PROGRAM PRG_LVCP5_Group3
VAR
    // Function Block Instance
    fbContactor: FB_ContactorControl;

    // Contactor 1 IO Structure  
    stContactor_IO: ST_ContactorIO;
    
    // Başlangıç konfigürasyonu için flag
    bContactorInitDone: BOOL := FALSE;
    bCapacitorInitDone: BOOL := FALSE;	
END_VAR



	M_Contactor();
	
	M_Capacitor();

METHOD M_Capacitor : BOOL
VAR
    nGroupIndex : INT;
END_VAR

nGroupIndex := 2;  // Grup 3 için index

IF NOT bCapacitorInitDone THEN
    // Grup 3 değerlerini ata
    GVL_LVCP5.astCompensationGroups[nGroupIndex].rPower := 10.0;
    GVL_LVCP5.astCompensationGroups[nGroupIndex].rVoltage := 450.0;
    GVL_LVCP5.astCompensationGroups[nGroupIndex].nQuantity := 8;
    GVL_LVCP5.astCompensationGroups[nGroupIndex].sTagPrefix := '+EP8-22C1';
    GVL_LVCP5.astCompensationGroups[nGroupIndex].sProductCode := 'ENT.CXD-450-10';
    
    bCapacitorInitDone := TRUE;
END_IF

// Grup 3 aktif durumu
GVL_LVCP5.abGroupActive[nGroupIndex] := stContactor_IO.bFeedback;

M_Capacitor := TRUE;
END_METHOD

METHOD M_Contactor : BOOL
VAR_INPUT
END_VAR
IF NOT bContactorInitDone THEN
    // Konfigürasyon parametreleri
    GVL_LVCP5.stGroup3_ContactorHMI.stConfig.sProjectCode := '+EP8-23K1';
    GVL_LVCP5.stGroup3_ContactorHMI.stConfig.sProductCode := 'SCH LC1G185LSEA';
    GVL_LVCP5.stGroup3_ContactorHMI.stConfig.rRatedCurrent := 185.0;
    GVL_LVCP5.stGroup3_ContactorHMI.stConfig.rRatedVoltage := 1000.0;
    GVL_LVCP5.stGroup3_ContactorHMI.stConfig.nPhaseCount := 3;
    GVL_LVCP5.stGroup3_ContactorHMI.stConfig.tFeedbackDelay := T#500MS;
    GVL_LVCP5.stGroup3_ContactorHMI.stConfig.tWeldedDelay := T#2S;
    GVL_LVCP5.stGroup3_ContactorHMI.stConfig.dwOperationLimit := 100000;
    
    // Başlangıç bakım sayacı
    GVL_LVCP5.stGroup3_ContactorHMI.stStatistics.dwRemainingOperations := GVL_LVCP5.stGroup3_ContactorHMI.stConfig.dwOperationLimit;
    
    bContactorInitDone := TRUE;
END_IF

// Function Block Çağrısı
fbContactor(
    // Fiziksel Girişler
    bFeedback 		:= stContactor_IO.bFeedback,
    bPLCControl 	:= stContactor_IO.bPLCControl,
    
    // Güvenlik Girişleri
    bSafetyLoop 	:= GVL_Alarm.bSafetyLoop,
    bInterlock 		:= FALSE,
    
    // Sistem Girişleri
    bMasterReset 	:= GVL_Alarm.bMasterReset,
    
    // HMI Bağlantısı
    stHMI 			:= GVL_LVCP5.stGroup3_ContactorHMI,
    
    // Fiziksel Çıkış
    bOutput 		=> stContactor_IO.bOutput
);

M_Contactor := TRUE;
END_METHOD

END_PROGRAM

(* stored: Version 1.1.0.1, ProductVersion 3.1.4024.15
   POU PRG_LVCP5_Group3: Id {38e6d7ac-9e59-4883-99aa-1c14646c4830}, SpecialFunc None
   Method M_Capacitor: Id {3e636123-f7be-49ee-97c3-ec5f67860945}
   Method M_Contactor: Id {a79b08c2-6da9-471f-aab8-bad4f25bcd6f} *)
